{attribute 'GeneratedUsingTerminal: KL8610-0005'}
{attribute addProperty BoxType "KL8610-0005"}
{attribute addProperty Id "KL8601_1AT %Q*KL_6576A6810KL8601_2AT %Q*KL_6576A6810KL8601_3AT %Q*KL_6576A6810KL8601_4AT %Q*KL_6576A6810KL8601_5AT %Q*KL_6576A6810KL8601_6AT %Q*KL_6576A6810"}
{attribute addProperty CRC "777836232"}
{attribute addProperty Size "0"}
TYPE KL_2E5CD6C8 :
STRUCT
	{attribute addProperty Name "KL8601_1"}
	KL8601_1 : KL_6576A681;
	{attribute addProperty Name "KL8601_2"}
	KL8601_2 : KL_6576A681;
	{attribute addProperty Name "KL8601_3"}
	KL8601_3 : KL_6576A681;
	{attribute addProperty Name "KL8601_4"}
	KL8601_4 : KL_6576A681;
	{attribute addProperty Name "KL8601_5"}
	KL8601_5 : KL_6576A681;
	{attribute addProperty Name "KL8601_6"}
	KL8601_6 : KL_6576A681;
END_STRUCT
END_TYPE

(* stored: Version 1.2.0.0, ProductVersion 3.1.4024.9
   DUT KL_2E5CD6C8: Id {8de2d57b-621a-4ba9-874a-c07c325d28de} *)
